DATA_BLOCK DB_DigInputOutput
STRUCT
    H_pos : BOOL;
    L_pos : BOOL;

    hoist_motor_on : BOOL;
    conveyor_motor_on : BOOL;
END_STRUCT
BEGIN


END_DATA_BLOCK
